(* Logix 5000 project; controller FF_Conveyors Emulate 5570 rev 20.11; software revision 20.04 *)

TASK MainTask (continuous, watchdog 500 ms) : MainProgram

MODULES
   Local : Emulate 5570 (ICP 3, rev 20.11)
      Digital_Input_1 : 1756-IB16 (ICP 1, rev 3.1, Input RPI 20 ms)
      Digital_Output_2 : vendor 1 type 7 code 16 (ICP 2, rev 3.1, Output RPI 20 ms)
END_MODULES

VAR_GLOBAL   (* controller tags *)
   B1_Fault : ALIAS FOR Local:1:I.Data.1;   // Belt 1 Faulted
   B1_Fault_ALM : BOOL;   // Belt 1 Fault Alarm
   B1_FTS_ALM : BOOL;   // Belt 1 Fail to Start Alarm
   B1_FTS_TMR : TIMER := (PRE := 2000);   // Belt 1 Fail to Start Timer
   B1_Run_CMD : ALIAS FOR Local:2:O.Data.0;   // Belt 1 Start Command
   B1_Running : ALIAS FOR Local:1:I.Data.0;   // Belt 1 Running
   B2_Fault : ALIAS FOR Local:1:I.Data.3;   // Belt 2 Faulted
   B2_Fault_ALM : BOOL;   // Belt 2 Fault Alarm
   B2_FTS_ALM : BOOL;   // Belt 2 Fail to Start Alarm
   B2_FTS_TMR : TIMER := (PRE := 2000);   // Belt 2 Fail to Start Timer
   B2_Run_CMD : ALIAS FOR Local:2:O.Data.1;   // Belt 2 Start Command
   B2_Running : ALIAS FOR Local:1:I.Data.2;   // Belt 2 Running
   B3_Fault : ALIAS FOR Local:1:I.Data.5;   // Belt 3 Faulted
   B3_Fault_ALM : BOOL;   // Belt 3 Fault Alarm
   B3_FTS_ALM : BOOL;   // Belt 3 Fail to Start Alarm
   B3_FTS_TMR : TIMER := (PRE := 2000);   // Belt 3 Fail to Start Timer
   B3_Run_CMD : ALIAS FOR Local:2:O.Data.2;   // Belt 3 Start Command
   B3_Running : ALIAS FOR Local:1:I.Data.4;   // Belt 3 Running
   B4_Fault : ALIAS FOR Local:1:I.Data.7;   // Belt 4 Faulted
   B4_Fault_ALM : BOOL;   // Belt 4 Fault Alarm
   B4_FTS_ALM : BOOL;   // Belt 4 Fail to Start Alarm
   B4_FTS_TMR : TIMER := (PRE := 2000);   // Belt 4 Fail to Start Timer
   B4_Run_CMD : ALIAS FOR Local:2:O.Data.3;   // Belt 4 Start Command
   B4_Running : ALIAS FOR Local:1:I.Data.6;   // Belt 4 Running
   B5_Fault : ALIAS FOR Local:1:I.Data.9;   // Belt 5 Faulted
   B5_Fault_ALM : BOOL;   // Belt 5 Fault Alarm
   B5_FTS_ALM : BOOL;   // Belt 5 Fail to Start Alarm
   B5_FTS_TMR : TIMER := (PRE := 2000);   // Belt 5 Fail to Start Alarm
   B5_Run_CMD : ALIAS FOR Local:2:O.Data.4;   // Belt 5 Start Command
   B5_Running : ALIAS FOR Local:1:I.Data.8;   // Belt 5 Running
END_VAR

PROGRAM MainProgram   (* main routine MainRoutine *)
VAR
   ALWAYS_OFF : BOOL;
   ALWAYS_ON : BOOL;
   B1_Auto_Start : BOOL;   // Belt 1 Auto Start 1 = ON, 0 = OFF
   B1_Man_Start : BOOL;   // Belt 1 Manual Start 1 = ON, 0 = OFF
   B1_RunTime : DINT;   // Belt 1 RunTime in Minutes
   B1_RunTime_RES : BOOL;   // Belt 1 Run Time Reset
   B1_RunTime_RTO : TIMER := (PRE := 60000);   // Belt 1 Run Time Timer
   B2_Auto_Start : BOOL;   // Belt 2 Auto Start 1 = ON, 0 = OFF
   B2_Man_Start : BOOL;   // Belt 2 Manual Start 1 = ON, 0 = OFF
   B2_RunTime : DINT;   // Belt 2 RunTime in Minutes
   B2_RunTime_RES : BOOL;   // Belt 2 Run Time Reset
   B2_RunTime_RTO : TIMER := (PRE := 60000);   // Belt 2 Run Time Timer
   B3_Auto_Start : BOOL;   // Belt 3 Auto Start 1 = ON, 0 = OFF
   B3_Man_Start : BOOL;   // Belt 3 Manual Start 1 = ON, 0 = OFF
   B3_RunTime : DINT;   // Belt 3 RunTime in Minutes
   B3_RunTime_RES : BOOL;   // Belt 3 Run Time Reset
   B3_RunTime_RTO : TIMER;   // Belt 3 Run Time Timer
   B4_Auto_Start : BOOL;   // Belt 4 Auto Start 1 = ON, 0 = OFF
   B4_Man_Start : BOOL;   // Belt 4 Manual Start 1 = ON, 0 = OFF
   B4_RunTime : DINT;   // Belt 4 RunTime in Minutes
   B4_RunTime_RES : BOOL;   // Belt 4 Run Time Reset
   B4_RunTime_RTO : TIMER;   // Belt 4 Run Time Timer
   B5_Auto_Start : BOOL;   // Belt 5 Manual Start 1 = ON, 0 = OFF
   B5_Man_Start : BOOL;   // Belt 5 Manual Start 1 = ON, 0 = OFF
   B5_RunTime_RES : BOOL;   // Belt 5 Run Time Reset
   B5_RunTime_RTO : TIMER;   // Belt 5 Run Time Timer
   DateTime : DINT[7];
   Global_ALM_RST : BOOL;   // Global Alarm Reset
   Seq_Step1_TMR : TIMER := (PRE := 1000);   // Sequence Step 1 Timer
   Sequence_Run : BOOL;   // Sequence Start 1 = Run, 0 = Stop
   Sequence_Start : BOOL;   // Sequence Start
   Sequence_Started : BOOL;   // Sequence Started
   Sequence_Stop : BOOL;   // Sequence Stop
   Sequence_Stopping : BOOL;   // Sequence Stopping
   Start_Seq_Step2_TMR : TIMER := (PRE := 1000);   // Start Sequence Step 2 Tmer
   Start_Seq_Step3_TMR : TIMER := (PRE := 1000);   // Start Sequence Step 3 Timer
   Start_Seq_Step4_TMR : TIMER := (PRE := 1000);   // Start Sequence Step 4 Timer
   Start_Seq_Step5_TMR : TIMER := (PRE := 1000);   // Start Sequence Step 5 Timer
   Stop_Seq_Step1_TMR : TIMER := (PRE := 1000);   // Stop Sequence Step 1 Timer
   Stop_Seq_Step2_TMR : TIMER := (PRE := 1000);   // Stop Sequence Step 2 Timer
   Stop_Seq_Step3_TMR : TIMER := (PRE := 1000);   // Stop Sequence Step 3 Timer
   Stop_Seq_Step4_TMR : TIMER := (PRE := 1000);   // Stop Sequence Step 4 Timer
   Stop_Seq_Step5_TMR : TIMER := (PRE := 1000);   // Stop Sequence Step 5 Timer
   System_MA : BOOL;   // System Manual/Auto Select 0=M, 1 = A
END_VAR

ROUTINE Belt_01   (* ladder *)
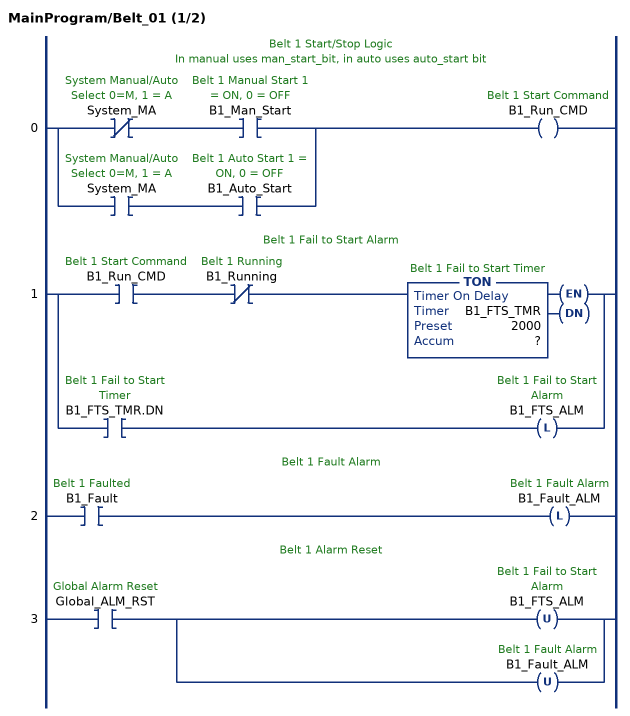
   // Belt 1 Start/Stop Logic
   // In manual uses man_start_bit, in auto uses auto_start bit
   0: [XIO(System_MA) XIC(B1_Man_Start) ,XIC(System_MA) XIC(B1_Auto_Start) ]OTE(B1_Run_CMD);
   // Belt 1 Fail to Start Alarm
   1: [XIC(B1_Run_CMD) XIO(B1_Running) TON(B1_FTS_TMR,?,?) ,XIC(B1_FTS_TMR.DN) OTL(B1_FTS_ALM) ];
   // Belt 1 Fault Alarm
   2: XIC(B1_Fault)OTL(B1_Fault_ALM);
   // Belt 1 Alarm Reset
   3: XIC(Global_ALM_RST)[OTU(B1_FTS_ALM) ,OTU(B1_Fault_ALM) ];
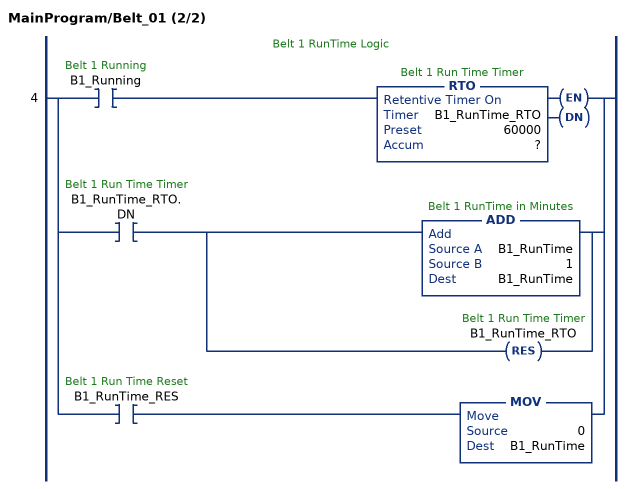
   // Belt 1 RunTime Logic
   4: [XIC(B1_Running) RTO(B1_RunTime_RTO,?,?) ,XIC(B1_RunTime_RTO.DN) [ADD(B1_RunTime,1,B1_RunTime) ,RES(B1_RunTime_RTO) ] ,XIC(B1_RunTime_RES) MOV(0,B1_RunTime) ];
END_ROUTINE

ROUTINE Belt_02   (* ladder *)
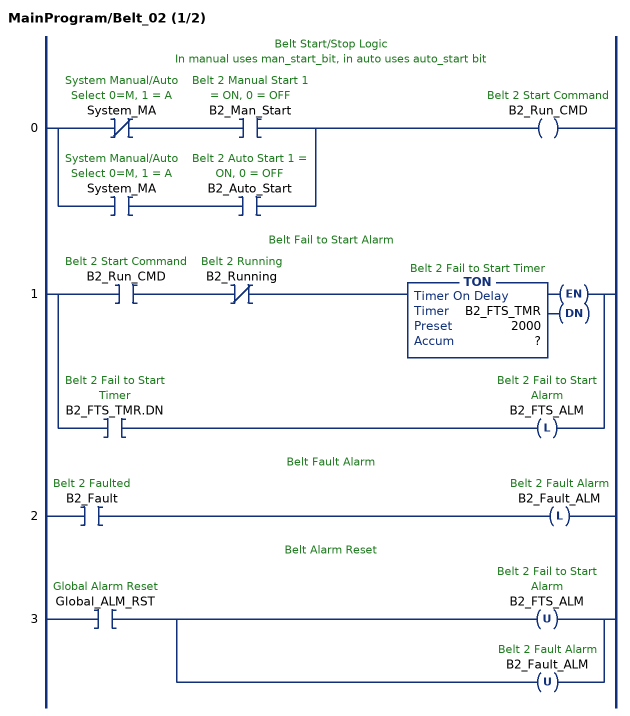
   // Belt Start/Stop Logic
   // In manual uses man_start_bit, in auto uses auto_start bit
   0: [XIO(System_MA) XIC(B2_Man_Start) ,XIC(System_MA) XIC(B2_Auto_Start) ]OTE(B2_Run_CMD);
   // Belt Fail to Start Alarm
   1: [XIC(B2_Run_CMD) XIO(B2_Running) TON(B2_FTS_TMR,?,?) ,XIC(B2_FTS_TMR.DN) OTL(B2_FTS_ALM) ];
   // Belt Fault Alarm
   2: XIC(B2_Fault)OTL(B2_Fault_ALM);
   // Belt Alarm Reset
   3: XIC(Global_ALM_RST)[OTU(B2_FTS_ALM) ,OTU(B2_Fault_ALM) ];
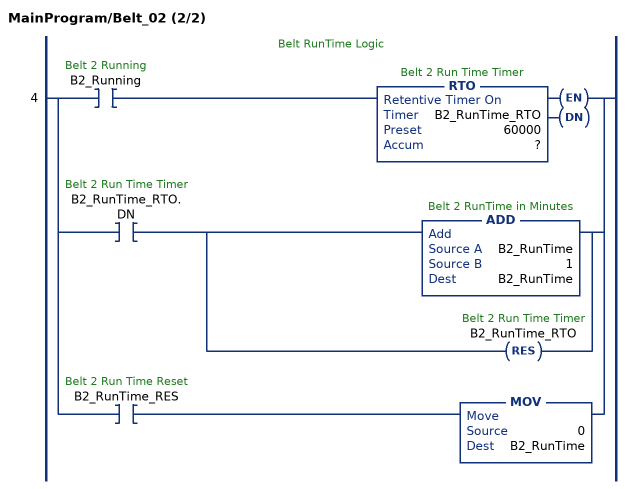
   // Belt RunTime Logic
   4: [XIC(B2_Running) RTO(B2_RunTime_RTO,?,?) ,XIC(B2_RunTime_RTO.DN) [ADD(B2_RunTime,1,B2_RunTime) ,RES(B2_RunTime_RTO) ] ,XIC(B2_RunTime_RES) MOV(0,B2_RunTime) ];
END_ROUTINE

ROUTINE Belt_03   (* ladder *)
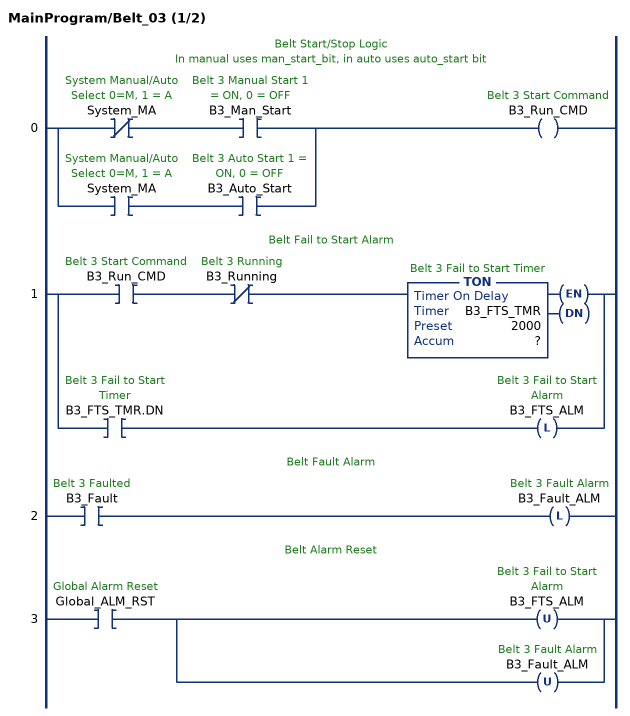
   // Belt Start/Stop Logic
   // In manual uses man_start_bit, in auto uses auto_start bit
   0: [XIO(System_MA) XIC(B3_Man_Start) ,XIC(System_MA) XIC(B3_Auto_Start) ]OTE(B3_Run_CMD);
   // Belt Fail to Start Alarm
   1: [XIC(B3_Run_CMD) XIO(B3_Running) TON(B3_FTS_TMR,?,?) ,XIC(B3_FTS_TMR.DN) OTL(B3_FTS_ALM) ];
   // Belt Fault Alarm
   2: XIC(B3_Fault)OTL(B3_Fault_ALM);
   // Belt Alarm Reset
   3: XIC(Global_ALM_RST)[OTU(B3_FTS_ALM) ,OTU(B3_Fault_ALM) ];
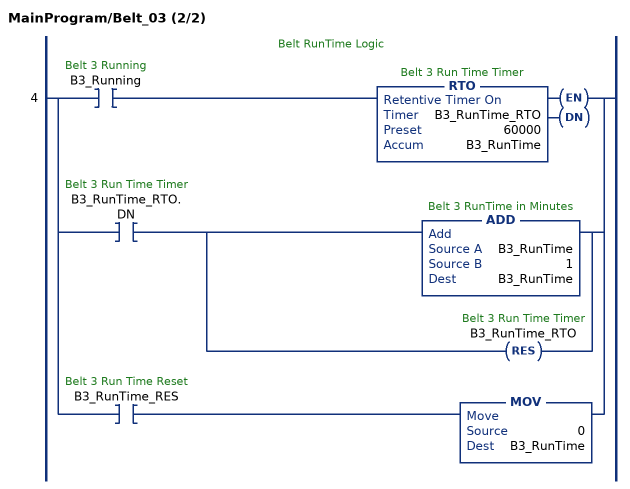
   // Belt RunTime Logic
   4: [XIC(B3_Running) RTO(B3_RunTime_RTO,60000,B3_RunTime) ,XIC(B3_RunTime_RTO.DN) [ADD(B3_RunTime,1,B3_RunTime) ,RES(B3_RunTime_RTO) ] ,XIC(B3_RunTime_RES) MOV(0,B3_RunTime) ];
END_ROUTINE

ROUTINE Belt_04   (* ladder *)
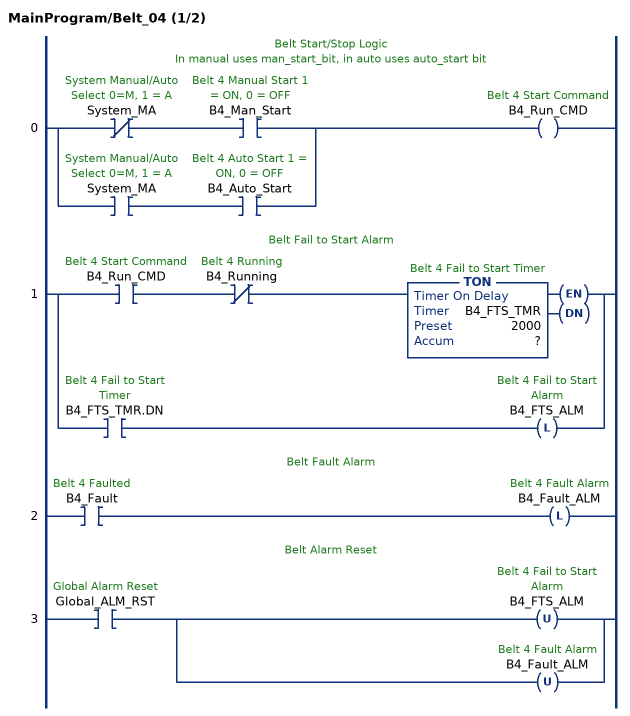
   // Belt Start/Stop Logic
   // In manual uses man_start_bit, in auto uses auto_start bit
   0: [XIO(System_MA) XIC(B4_Man_Start) ,XIC(System_MA) XIC(B4_Auto_Start) ]OTE(B4_Run_CMD);
   // Belt Fail to Start Alarm
   1: [XIC(B4_Run_CMD) XIO(B4_Running) TON(B4_FTS_TMR,?,?) ,XIC(B4_FTS_TMR.DN) OTL(B4_FTS_ALM) ];
   // Belt Fault Alarm
   2: XIC(B4_Fault)OTL(B4_Fault_ALM);
   // Belt Alarm Reset
   3: XIC(Global_ALM_RST)[OTU(B4_FTS_ALM) ,OTU(B4_Fault_ALM) ];
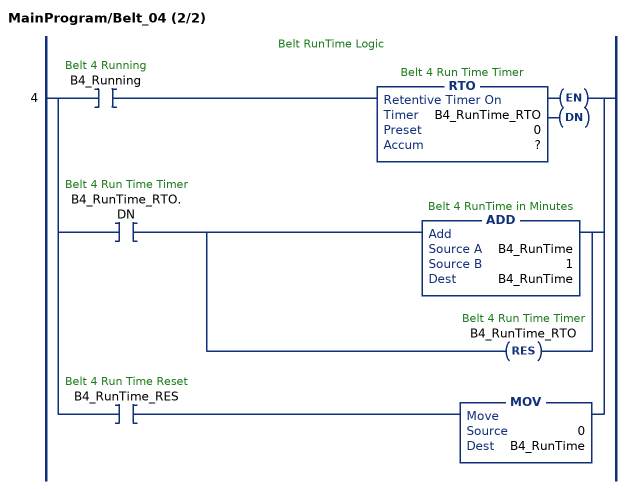
   // Belt RunTime Logic
   4: [XIC(B4_Running) RTO(B4_RunTime_RTO,?,?) ,XIC(B4_RunTime_RTO.DN) [ADD(B4_RunTime,1,B4_RunTime) ,RES(B4_RunTime_RTO) ] ,XIC(B4_RunTime_RES) MOV(0,B4_RunTime) ];
END_ROUTINE

ROUTINE Belt_05   (* ladder *)
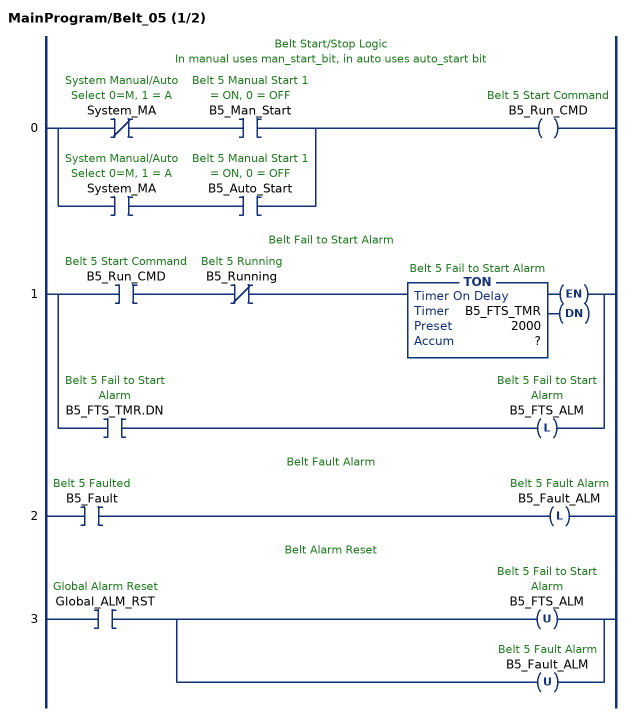
   // Belt Start/Stop Logic
   // In manual uses man_start_bit, in auto uses auto_start bit
   0: [XIO(System_MA) XIC(B5_Man_Start) ,XIC(System_MA) XIC(B5_Auto_Start) ]OTE(B5_Run_CMD);
   // Belt Fail to Start Alarm
   1: [XIC(B5_Run_CMD) XIO(B5_Running) TON(B5_FTS_TMR,?,?) ,XIC(B5_FTS_TMR.DN) OTL(B5_FTS_ALM) ];
   // Belt Fault Alarm
   2: XIC(B5_Fault)OTL(B5_Fault_ALM);
   // Belt Alarm Reset
   3: XIC(Global_ALM_RST)[OTU(B5_FTS_ALM) ,OTU(B5_Fault_ALM) ];
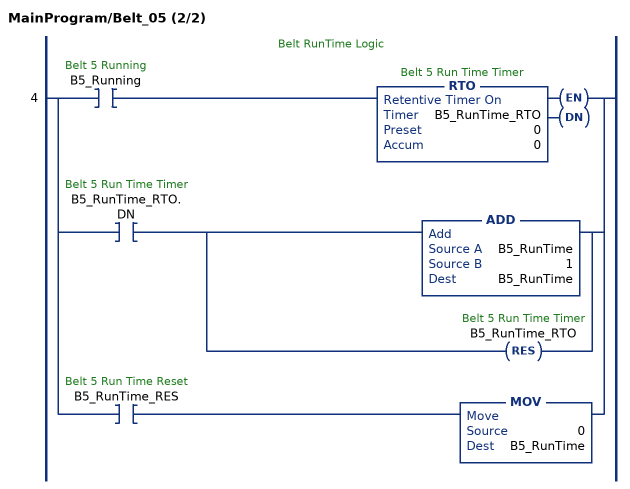
   // Belt RunTime Logic
   4: [XIC(B5_Running) RTO(B5_RunTime_RTO,0,0) ,XIC(B5_RunTime_RTO.DN) [ADD(B5_RunTime,1,B5_RunTime) ,RES(B5_RunTime_RTO) ] ,XIC(B5_RunTime_RES) MOV(0,B5_RunTime) ];
END_ROUTINE

ROUTINE MainRoutine   (* ladder *)
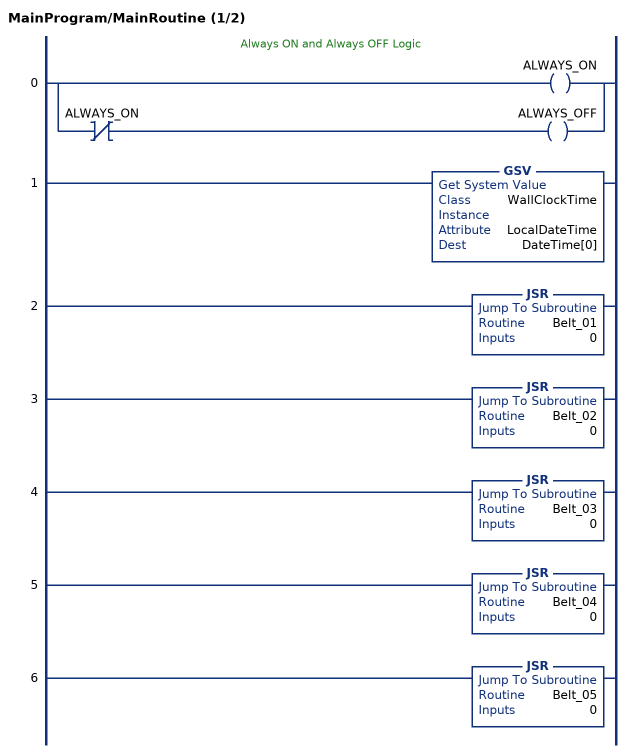
   // Always ON and Always OFF Logic
   0: [OTE(ALWAYS_ON) ,XIO(ALWAYS_ON) OTE(ALWAYS_OFF) ];
   1: GSV(WallClockTime,,LocalDateTime,DateTime[0]);
   2: JSR(Belt_01,0);
   3: JSR(Belt_02,0);
   4: JSR(Belt_03,0);
   5: JSR(Belt_04,0);
   6: JSR(Belt_05,0);
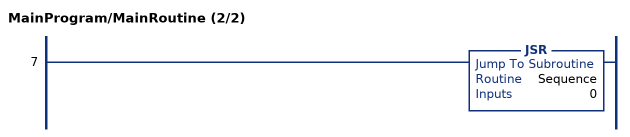
   7: JSR(Sequence,0);
END_ROUTINE

ROUTINE Sequence   (* ladder *)
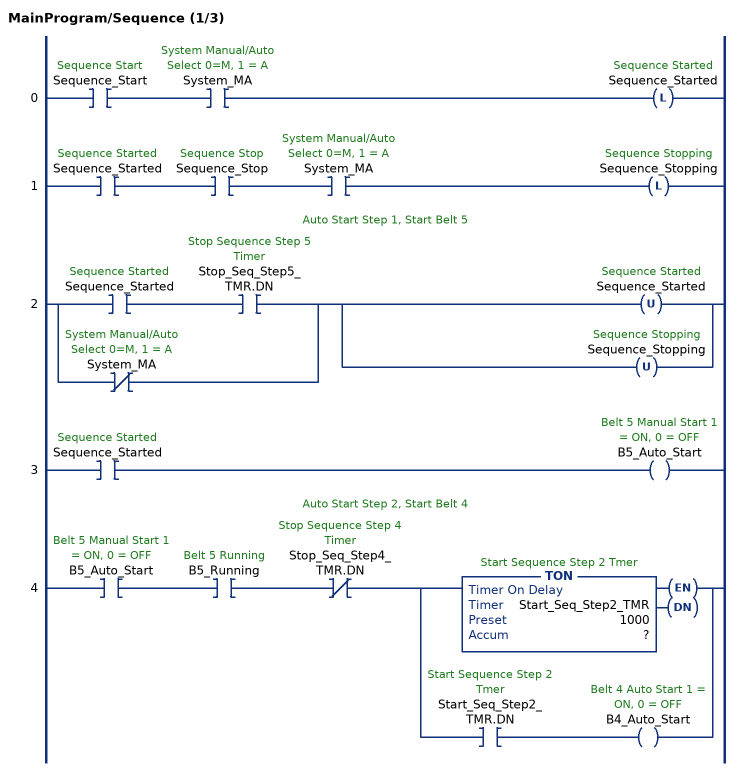
   0: XIC(Sequence_Start)XIC(System_MA)OTL(Sequence_Started);
   1: XIC(Sequence_Started)XIC(Sequence_Stop)XIC(System_MA)OTL(Sequence_Stopping);
   // Auto Start Step 1, Start Belt 5
   2: [XIC(Sequence_Started) XIC(Stop_Seq_Step5_TMR.DN) ,XIO(System_MA) ][OTU(Sequence_Started) ,OTU(Sequence_Stopping) ];
   3: XIC(Sequence_Started)OTE(B5_Auto_Start);
   // Auto Start Step 2, Start Belt 4
   4: XIC(B5_Auto_Start)XIC(B5_Running)XIO(Stop_Seq_Step4_TMR.DN)[TON(Start_Seq_Step2_TMR,?,?) ,XIC(Start_Seq_Step2_TMR.DN) OTE(B4_Auto_Start) ];
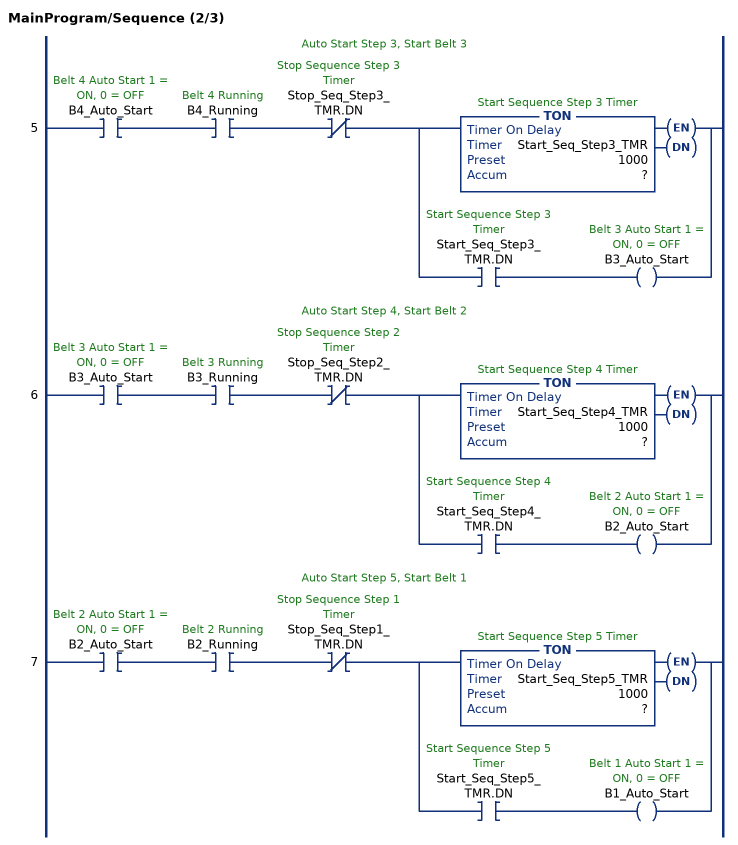
   // Auto Start Step 3, Start Belt 3
   5: XIC(B4_Auto_Start)XIC(B4_Running)XIO(Stop_Seq_Step3_TMR.DN)[TON(Start_Seq_Step3_TMR,?,?) ,XIC(Start_Seq_Step3_TMR.DN) OTE(B3_Auto_Start) ];
   // Auto Start Step 4, Start Belt 2
   6: XIC(B3_Auto_Start)XIC(B3_Running)XIO(Stop_Seq_Step2_TMR.DN)[TON(Start_Seq_Step4_TMR,?,?) ,XIC(Start_Seq_Step4_TMR.DN) OTE(B2_Auto_Start) ];
   // Auto Start Step 5, Start Belt 1
   7: XIC(B2_Auto_Start)XIC(B2_Running)XIO(Stop_Seq_Step1_TMR.DN)[TON(Start_Seq_Step5_TMR,?,?) ,XIC(Start_Seq_Step5_TMR.DN) OTE(B1_Auto_Start) ];
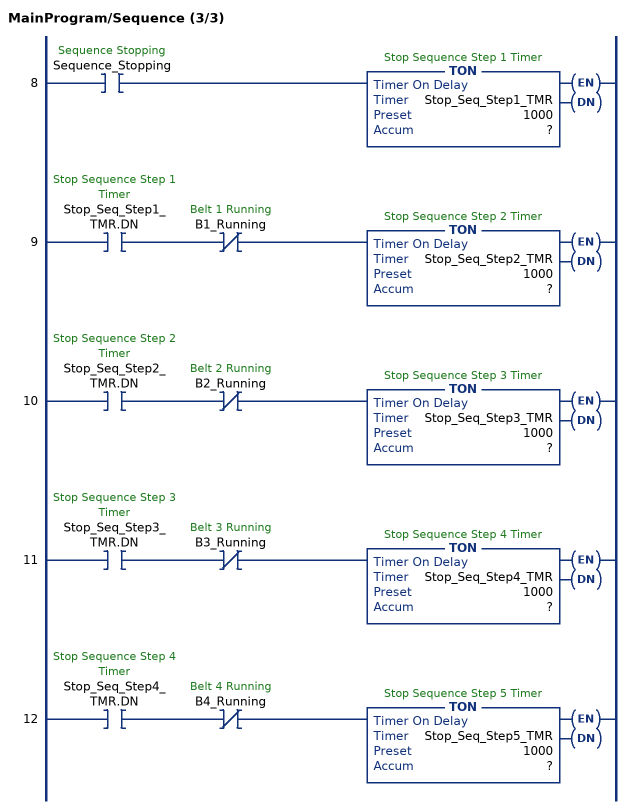
   8: XIC(Sequence_Stopping)TON(Stop_Seq_Step1_TMR,?,?);
   9: XIC(Stop_Seq_Step1_TMR.DN)XIO(B1_Running)TON(Stop_Seq_Step2_TMR,?,?);
   10: XIC(Stop_Seq_Step2_TMR.DN)XIO(B2_Running)TON(Stop_Seq_Step3_TMR,?,?);
   11: XIC(Stop_Seq_Step3_TMR.DN)XIO(B3_Running)TON(Stop_Seq_Step4_TMR,?,?);
   12: XIC(Stop_Seq_Step4_TMR.DN)XIO(B4_Running)TON(Stop_Seq_Step5_TMR,?,?);
END_ROUTINE
END_PROGRAM
